PROGRAM GCC2
VAR
	rfbAdsRead: ADSREAD;
	sNetId: T_AmsNetID:='192.168.0.3';
	sPort: T_AmsPort:=851;
	bRead:BOOL;
	r_Press :REAL;
END_VAR

rfbAdsRead(
	NETID:= sNetID , 
	PORT:= sPort, 
	IDXGRP:= 16#4040, 
	IDXOFFS:= 971076 , 
	LEN:= SIZEOF(r_Press), 
	DESTADDR:= ADR(r_Press) , 
	READ:= bRead);

END_PROGRAM

(* stored: Version 1.1.0.1, ProductVersion 3.1.4022.3
   POU GCC2: Id {0d92b97a-0c10-46eb-9d94-2022c80c6ed6}, SpecialFunc None *)
